ABB RAPID module: Parameters.mod

MODULE Parameters


!************************************************************************************************!
!********************ABB **************************!
  VAR string server_socket_IP:="192.168.11.101";   !***** ABB controller WAN IP  "192.168.0.1"
  VAR num host_prot:=2000;                      !***** prot

!************************************************************************************************!
!**********************************************!
const stoppointdata my_inpos := [ inpos, TRUE, [ 0, 0, 0.1, 5], 0, 0, "", 0, 0];!******
const speeddata my_speed := [ 10000, 4000, 3400, 1800 ];!**********my_speed:

VAR zonedata my_path := [ FALSE, 25, 40, 40, 10, 35, 5 ];!*******TCP

!VAR speeddata my_init_speed := [ 50, 10, 20, 5 ];
VAR speeddata my_init_speed := [ 30, 30, 20, 5 ];
VAR speeddata g_SpeedRun;

VAR robtarget palletA_Col;
VAR robtarget palletA_Row;
VAR robtarget palletB_Col;
VAR robtarget palletB_Row;
VAR robtarget point_GetCoilCurrPot;
VAR num Snap:=0;
var num rUdisp;
VAR num i;


!************************************************************************************************!
!**********************************************!
CONST num Order_Otr_Num:=9;

VAR num RobotLmtZ:=185;
VAR num SafeLmtZ:=185;
!************************************************************************************************!

VAR num g_DryRun;
var num g_NextGet;
!************************************************************************************************!
!************************************************************************************************!
!************************************************************************************************!
!************************************************************************************************!
!************************************************************************************************!
PERS string TodayDate:="2020-04-08";

ENDMODULE
